// Mitsubishi GX Works2 project: 자동화실린더   PLC: Q02/Q02H

PROGRAM MAIN
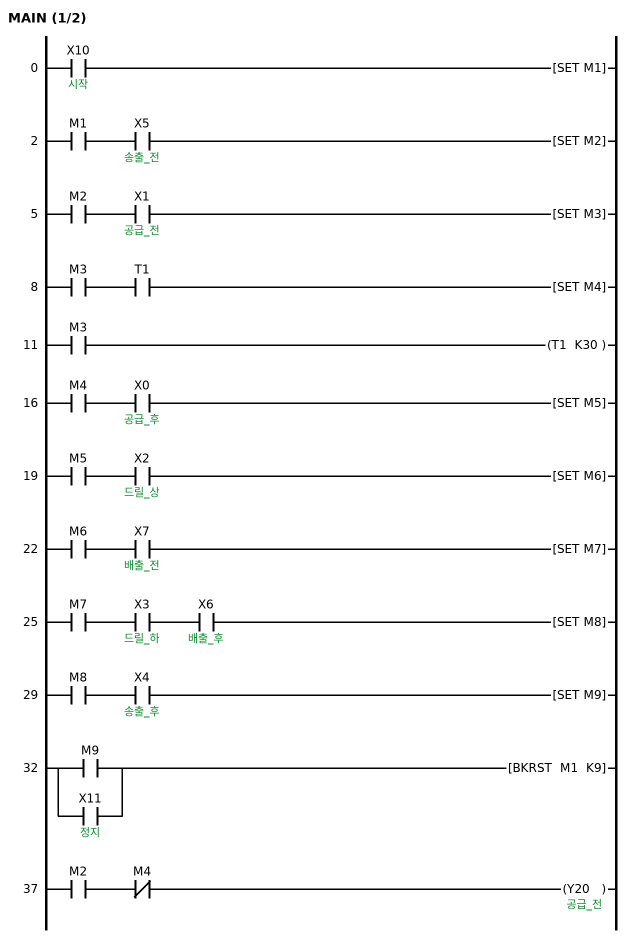
0     LD      X10  ; 시작
      SET     M1
2     LD      M1
      AND     X5  ; 송출_전
      SET     M2
5     LD      M2
      AND     X1  ; 공급_전
      SET     M3
8     LD      M3
      AND     T1
      SET     M4
11    LD      M3
      OUT     T1 K30
16    LD      M4
      AND     X0  ; 공급_후
      SET     M5
19    LD      M5
      AND     X2  ; 드릴_상
      SET     M6
22    LD      M6
      AND     X7  ; 배출_전
      SET     M7
25    LD      M7
      AND     X3  ; 드릴_하
      AND     X6  ; 배출_후
      SET     M8
29    LD      M8
      AND     X4  ; 송출_후
      SET     M9
32    LD      M9
      OR      X11  ; 정지
      BKRST   M1 K9
37    LD      M2
      ANI     M4
      OUT     Y20  ; 공급_전
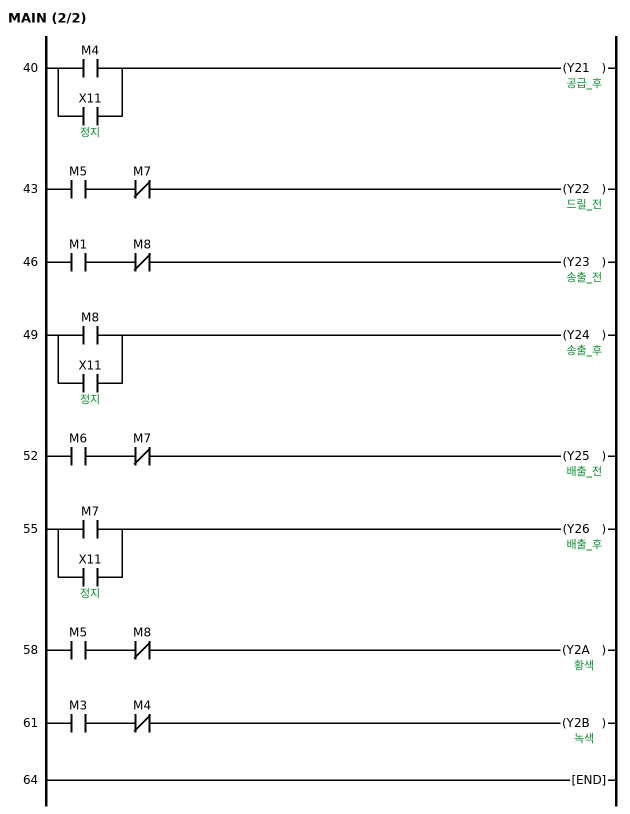
40    LD      M4
      OR      X11  ; 정지
      OUT     Y21  ; 공급_후
43    LD      M5
      ANI     M7
      OUT     Y22  ; 드릴_전
46    LD      M1
      ANI     M8
      OUT     Y23  ; 송출_전
49    LD      M8
      OR      X11  ; 정지
      OUT     Y24  ; 송출_후
52    LD      M6
      ANI     M7
      OUT     Y25  ; 배출_전
55    LD      M7
      OR      X11  ; 정지
      OUT     Y26  ; 배출_후
58    LD      M5
      ANI     M8
      OUT     Y2A  ; 황색
61    LD      M3
      ANI     M4
      OUT     Y2B  ; 녹색
64    END
END_PROGRAM

// device comments not shown above
X8  ; 메거진
X9  ; 비금속
X0A  ; 금속
Y27  ; 컨베어
Y28  ; 가공드
Y29  ; 적색
